(* Logix 5000 project; controller cal1615 1756-L62 rev 20.19; software revision 20.05; part 81 of 81 *)
(* tags used below, declared in another part *)
   A00 : ALIAS FOR hmi_dint[0].0;
   A12 : ALIAS FOR hmi_dint[0].12;
   A30 : ALIAS FOR hmi_dint[0].30;
   acc_settle_tmr : TIMER;
   acc_taper : REAL;
   add_sys_ramp : sys_Ramp;   // Addon Ramp
   ai_lpt01_pct : REAL;   // AI: Linear Position Transducer [%]
   ao_prs01 : REAL;   // AO: Pressure 1
   ao_prs02 : REAL;   // AO: Pressure 2
   control_to_empty : ALIAS FOR hmi_dint[9].13;
   di_ss_close_nip : ALIAS FOR p00_io_winder:5:I.14;
   di_ss_nip_auto : ALIAS FOR p00_io_winder:5:I.13;
   do_carriage_lift_sol : ALIAS FOR p00_io_winder:4:O.7;
   do_close_nip_sol : ALIAS FOR p00_io_winder:4:O.8;
   do_nip_illuminated_ss : ALIAS FOR p00_io_winder:4:O.6;
   enable_control : BOOL;   // Accumulator - Enable Control
   Me : ALIAS FOR p00_wac;
   nip_auto_open_request : BOOL;   // Nip Auto Open Request
   nip_close_request : ALIAS FOR hmi_dint[9].7;
   nip_mode_auto : BOOL;   // Nip Mode Auto
   nip_open_dwell : TIMER;   // Nip Roll Open Dwell Payout must be established before the nip lets go
   nip_open_request : BOOL;   // Nip Open Request
   nip_open_selected : BOOL;   // Nip Selector in OPEN Neither Auto nor Close
   oneshot : DINT;
   p00_wac_speed_offset : REAL;
   param_acc_capacity_ft : REAL;   // Parameter Accumulator Web Capacity at Full Stroke 26 s at 23 fpm measured [ft]
   param_acc_empty_hyst : REAL;
   param_acc_empty_pct : REAL;
   param_acc_min_limit : REAL;   // Parameter Accumulator Low Min Limimt
   param_acc_settle_ms : DINT;
   param_acc_taper_pct : REAL;
   param_accel_rate : REAL;   // Parameter Acceleration Rate
   param_counter_prs : REAL;   // Parameter Counter Pressure
   param_decel_rate : REAL;   // Parameter Decleration Rate
   param_payout_overspeed : REAL;
   param_prs_empty : REAL;
   param_prs_fill : REAL;
   param_prs_payout : REAL;
   pb_acc_on : ALIAS FOR hmi_dint[9].2;
   request_fill : ALIAS FOR hmi_dint[9].1;
   selected_pressure : REAL;   // Accumulator Selected Tension Pressure
   timer_nip_open_delay : TIMER;   // Nip Open Dwell Timer
   W00 : ALIAS FOR hmi_dint[2].0;
   FAULT : BOOL;   // Fault AFI
   HMI : BOOL;   // AFI HMI
   nip_mode_close : BOOL;   // Nip Mode Close
   p00_FlashBit_1Sec : BOOL;   // System Flash Bit 1 Second
   p00_pb_lamp_test : BOOL;
   p00_wac : Accumulator;   // Winder Accumulator
   p00_wac_enabled : BOOL;   // Winder Accumulator Enabled Carriage lift on and pressure commanded Controls which loop holds web tension
   p00_wac_position_pct : REAL;   // Winder Accumulator Carriage Position Filtered [% of Stroke]
   p00_wac_settled : BOOL;
   p01r02_plc_scan_time_in_sec : REAL;   // System PLC Scan Time in Seconds
   p01r09 : routine;   // System Modes
   p01r12_zero_line_speed : BOOL;   // System Line Accel Decel Control Line Speed at Zero
   p29r15_request_run : BOOL;   // Winder Winder A VFD Request Run
   p29r16_request_run : BOOL;   // Winder Winder B VFD Request Run
(* P31_WAC, continued *)

ROUTINE R11_Modes   (* ladder *)
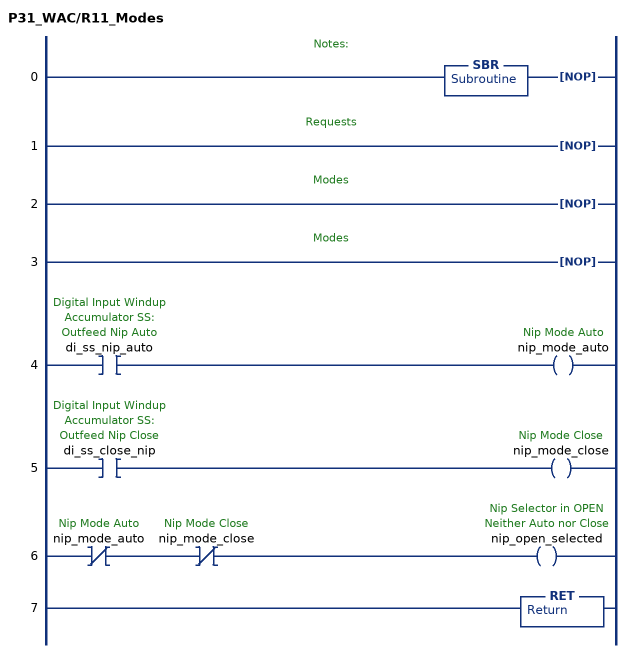
   // Notes:
   0: SBR()NOP();
   // Requests
   1: NOP();
   // Modes
   2: NOP();
   // Modes
   3: NOP();
   4: XIC(di_ss_nip_auto)OTE(nip_mode_auto);
   5: XIC(di_ss_close_nip)OTE(nip_mode_close);
   6: XIO(nip_mode_auto)XIO(nip_mode_close)OTE(nip_open_selected);
   7: RET();
END_ROUTINE

ROUTINE R21_Fill_Request   (* ladder *)
// WAC
// Fill Request and Tension Enable
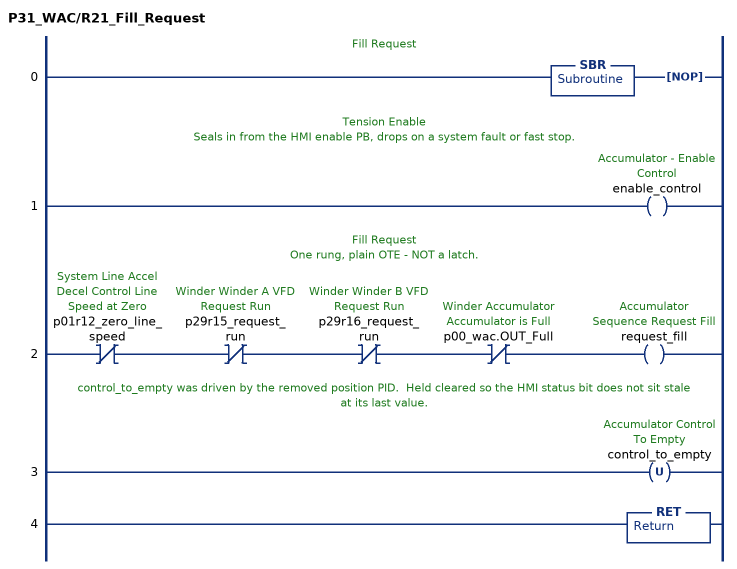
   // Fill Request
   0: SBR()NOP();
   // Tension Enable
   // Seals in from the HMI enable PB, drops on a system fault or fast stop.
   1: OTE(enable_control);
   // Fill Request
   // One rung, plain OTE - NOT a latch.
   2: XIO(p01r12_zero_line_speed)XIO(p29r15_request_run)XIO(p29r16_request_run)XIO(p00_wac.OUT_Full)OTE(request_fill);
   // control_to_empty was driven by the removed position PID.  Held cleared so the HMI status bit does not sit stale at its last value.
   3: OTU(control_to_empty);
   4: RET();
END_ROUTINE

ROUTINE R22_Fill_Pressure   (* ladder *)
// Windup Accumulator
// Fill Pressure
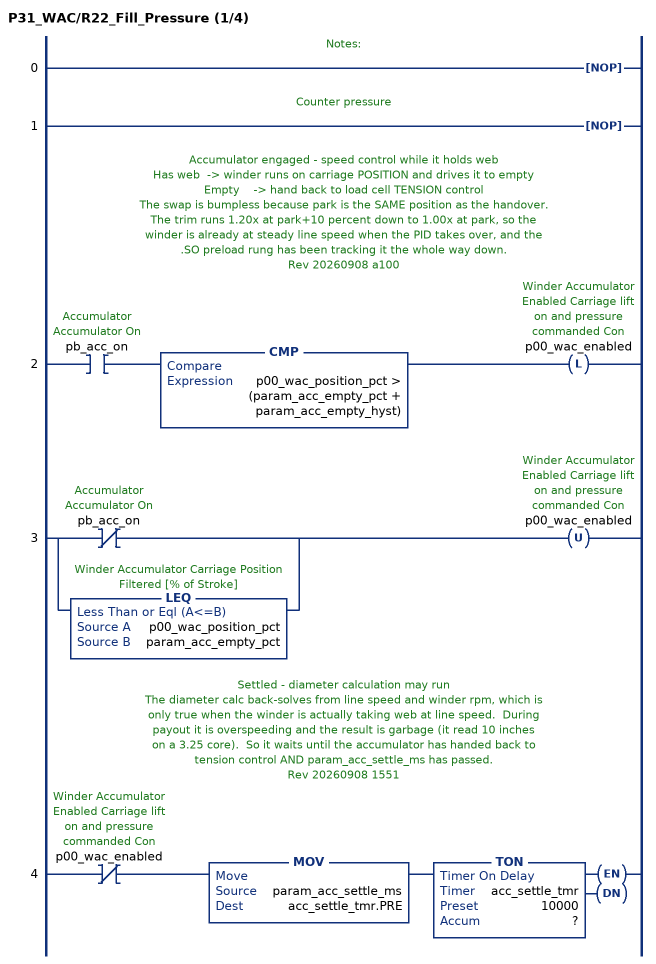
   // Notes:
   0: NOP();
   // Counter pressure
   1: NOP();
   // Accumulator engaged - speed control while it holds web
   // Has web  -> winder runs on carriage POSITION and drives it to empty
   // Empty    -> hand back to load cell TENSION control
   // The swap is bumpless because park is the SAME position as the handover.
   // The trim runs 1.20x at park+10 percent down to 1.00x at park, so the
   // winder is already at steady line speed when the PID takes over, and the
   // .SO preload rung has been tracking it the whole way down.
   // Rev 20260908 a100
   2: XIC(pb_acc_on)CMP(p00_wac_position_pct > (param_acc_empty_pct + param_acc_empty_hyst))OTL(p00_wac_enabled);
   3: [XIO(pb_acc_on) ,LEQ(p00_wac_position_pct,param_acc_empty_pct) ]OTU(p00_wac_enabled);
   // Settled - diameter calculation may run
   // The diameter calc back-solves from line speed and winder rpm, which is
   // only true when the winder is actually taking web at line speed.  During
   // payout it is overspeeding and the result is garbage (it read 10 inches
   // on a 3.25 core).  So it waits until the accumulator has handed back to
   // tension control AND param_acc_settle_ms has passed.
   // Rev 20260908 1551
   4: XIO(p00_wac_enabled)MOV(param_acc_settle_ms,acc_settle_tmr.PRE)TON(acc_settle_tmr,?,?);
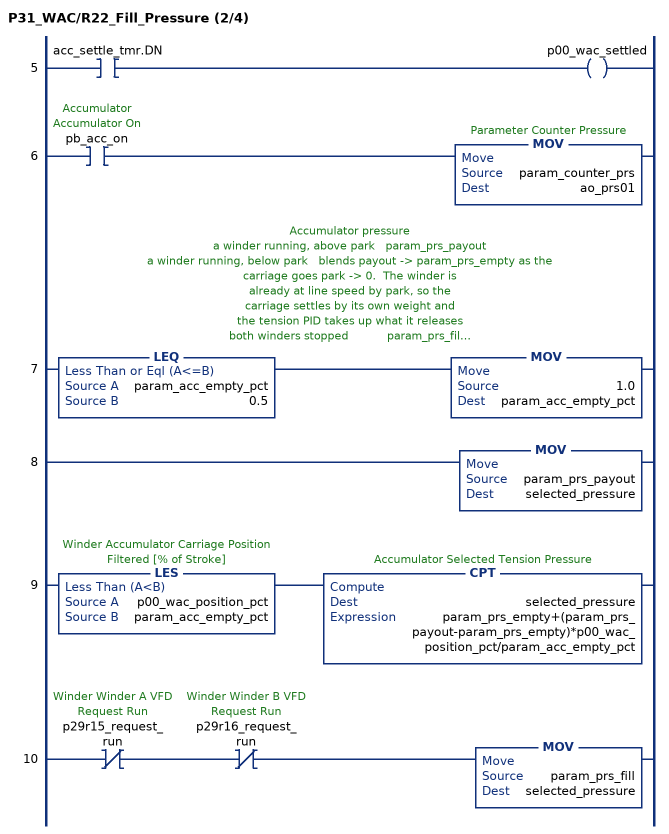
   5: XIC(acc_settle_tmr.DN)OTE(p00_wac_settled);
   6: XIC(pb_acc_on)MOV(param_counter_prs,ao_prs01);
   // Accumulator pressure
   //   a winder running, above park   param_prs_payout
   //   a winder running, below park   blends payout -> param_prs_empty as the
   //                                  carriage goes park -> 0.  The winder is
   //                                  already at line speed by park, so the
   //                                  carriage settles by its own weight and
   //                                  the tension PID takes up what it releases
   //   both winders stopped           param_prs_fill
   // sys_Ramp below smooths every change.
   // Rev 20260908 1551
   7: LEQ(param_acc_empty_pct,0.5)MOV(1.0,param_acc_empty_pct);
   8: MOV(param_prs_payout,selected_pressure);
   9: LES(p00_wac_position_pct,param_acc_empty_pct)CPT(selected_pressure,param_prs_empty+(param_prs_payout-param_prs_empty)*p00_wac_position_pct/param_acc_empty_pct);
   10: XIO(p29r15_request_run)XIO(p29r16_request_run)MOV(param_prs_fill,selected_pressure);
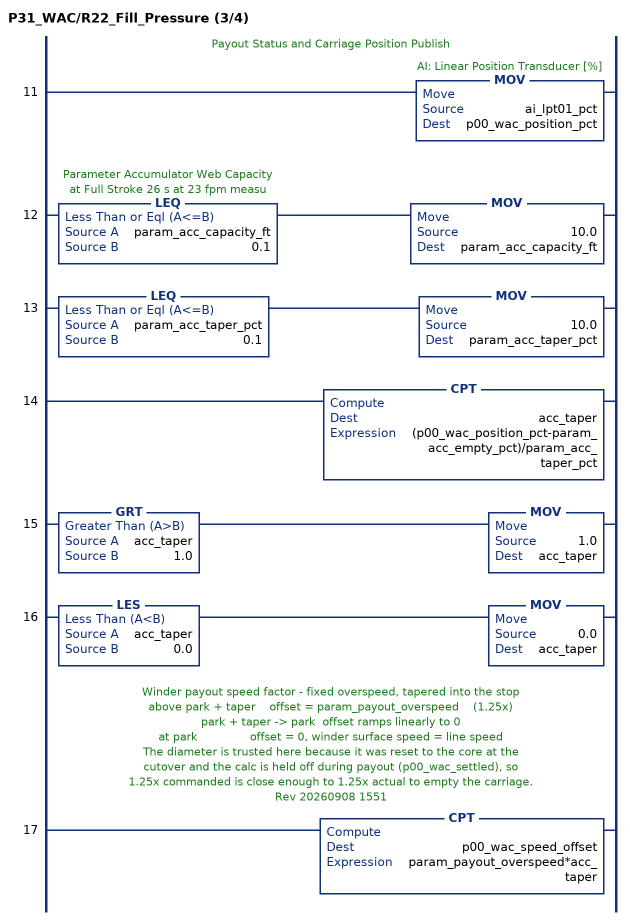
   // Payout Status and Carriage Position Publish
   11: MOV(ai_lpt01_pct,p00_wac_position_pct);
   12: LEQ(param_acc_capacity_ft,0.1)MOV(10.0,param_acc_capacity_ft);
   13: LEQ(param_acc_taper_pct,0.1)MOV(10.0,param_acc_taper_pct);
   14: CPT(acc_taper,(p00_wac_position_pct-param_acc_empty_pct)/param_acc_taper_pct);
   15: GRT(acc_taper,1.0)MOV(1.0,acc_taper);
   16: LES(acc_taper,0.0)MOV(0.0,acc_taper);
   // Winder payout speed factor - fixed overspeed, tapered into the stop
   //   above park + taper    offset = param_payout_overspeed    (1.25x)
   //   park + taper -> park  offset ramps linearly to 0
   //   at park               offset = 0, winder surface speed = line speed
   // The diameter is trusted here because it was reset to the core at the
   // cutover and the calc is held off during payout (p00_wac_settled), so
   // 1.25x commanded is close enough to 1.25x actual to empty the carriage.
   // Rev 20260908 1551
   17: CPT(p00_wac_speed_offset,param_payout_overspeed*acc_taper);
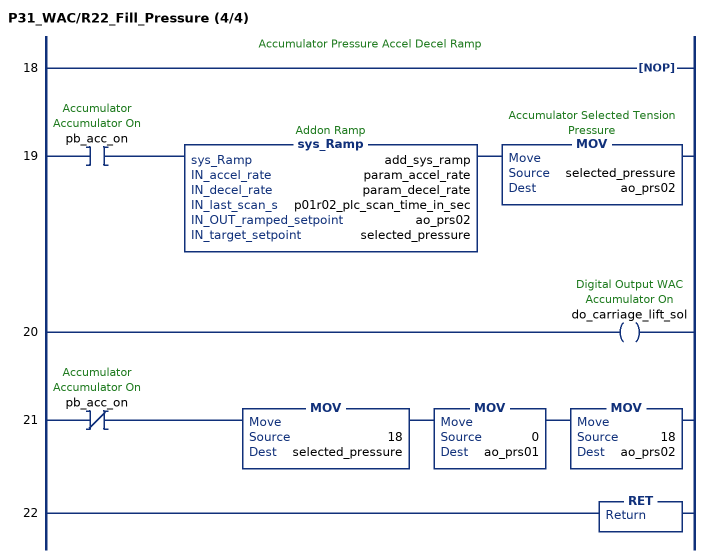
   // Accumulator Pressure Accel Decel Ramp
   18: NOP();
   19: XIC(pb_acc_on)sys_Ramp(add_sys_ramp,param_accel_rate,param_decel_rate,p01r02_plc_scan_time_in_sec,ao_prs02,selected_pressure)MOV(selected_pressure,ao_prs02);
   20: OTE(do_carriage_lift_sol);
   21: XIO(pb_acc_on)MOV(18,selected_pressure)MOV(0,ao_prs01)MOV(18,ao_prs02);
   22: RET();
END_ROUTINE

ROUTINE R31_Nip_Roll   (* ladder *)
// WAC
// Nip Roll
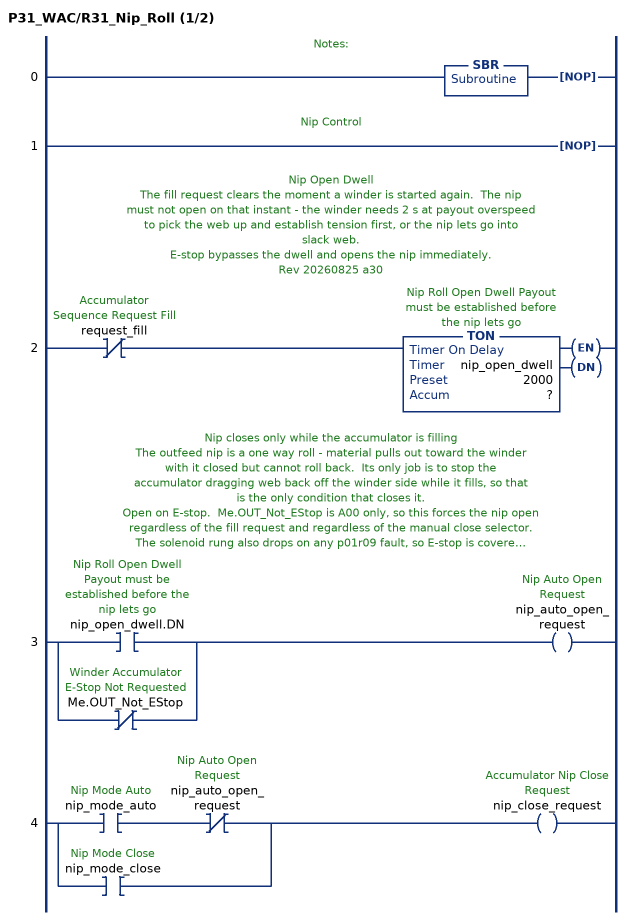
   // Notes:
   0: SBR()NOP();
   // Nip Control
   1: NOP();
   // Nip Open Dwell
   // The fill request clears the moment a winder is started again.  The nip
   // must not open on that instant - the winder needs 2 s at payout overspeed
   // to pick the web up and establish tension first, or the nip lets go into
   // slack web.
   // E-stop bypasses the dwell and opens the nip immediately.
   // Rev 20260825 a30
   2: XIO(request_fill)TON(nip_open_dwell,?,?);
   // Nip closes only while the accumulator is filling
   // The outfeed nip is a one way roll - material pulls out toward the winder
   // with it closed but cannot roll back.  Its only job is to stop the
   // accumulator dragging web back off the winder side while it fills, so that
   // is the only condition that closes it.
   // Open on E-stop.  Me.OUT_Not_EStop is A00 only, so this forces the nip open
   // regardless of the fill request and regardless of the manual close selector.
   // The solenoid rung also drops on any p01r09 fault, so E-stop is covered
   // twice - deliberately.
   // Previously opened on accumulator level above param_acc_min_limit.  That
   // left it open during the fill, which is the one time it needs to be shut.
   // No open delay - the level-based version needed one, this does not.
   // timer_nip_open_delay is left declared and unused.
   // Rev 20260825 a12
   3: [XIC(nip_open_dwell.DN) ,XIO(Me.OUT_Not_EStop) ]OTE(nip_auto_open_request);
   4: [XIC(nip_mode_auto) XIO(nip_auto_open_request) ,XIC(nip_mode_close) ]OTE(nip_close_request);
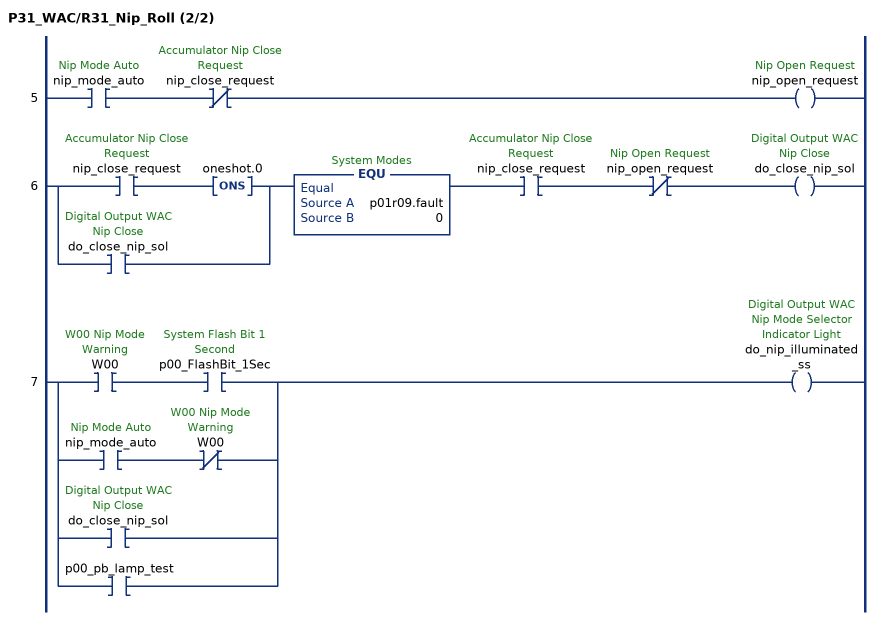
   5: XIC(nip_mode_auto)XIO(nip_close_request)OTE(nip_open_request);
   6: [XIC(nip_close_request) ONS(oneshot.0) ,XIC(do_close_nip_sol) ]EQU(p01r09.fault,0)XIC(nip_close_request)XIO(nip_open_request)OTE(do_close_nip_sol);
   7: [XIC(W00) XIC(p00_FlashBit_1Sec) ,XIC(nip_mode_auto) XIO(W00) ,XIC(do_close_nip_sol) ,XIC(p00_pb_lamp_test) ]OTE(do_nip_illuminated_ss);
END_ROUTINE
END_PROGRAM

PROGRAM ZZZ
END_PROGRAM
